SUBAPPLICATION Automatik_aus (* Subapplication Type *)
  (* Standard: 61499-2 *)
  (* Version 1.0, 2023-02-07, franz *)
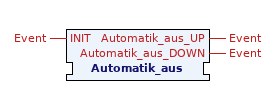
  EVENT_INPUT
    INIT;
  END_EVENT
  EVENT_OUTPUT
    Automatik_aus_UP;
    Automatik_aus_DOWN;
  END_EVENT
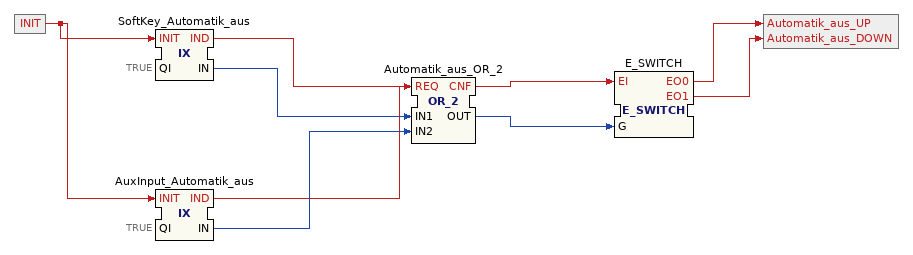
  FBS
    SoftKey_Automatik_aus : IX(QI := TRUE);
    AuxInput_Automatik_aus : IX(QI := TRUE);
    Automatik_aus_OR_2 : OR_2;
    E_SWITCH : E_SWITCH;
  END_FBS
  EVENT_CONNECTIONS
    INIT TO SoftKey_Automatik_aus.INIT;
    INIT TO AuxInput_Automatik_aus.INIT;
    SoftKey_Automatik_aus.IND TO Automatik_aus_OR_2.REQ;
    AuxInput_Automatik_aus.IND TO Automatik_aus_OR_2.REQ;
    Automatik_aus_OR_2.CNF TO E_SWITCH.EI;
    E_SWITCH.EO0 TO Automatik_aus_UP;
    E_SWITCH.EO1 TO Automatik_aus_DOWN;
  END_CONNECTIONS
  DATA_CONNECTIONS
    SoftKey_Automatik_aus.IN TO Automatik_aus_OR_2.IN1;
    AuxInput_Automatik_aus.IN TO Automatik_aus_OR_2.IN2;
    Automatik_aus_OR_2.OUT TO E_SWITCH.G;
  END_CONNECTIONS
END_SUBAPPLICATION
